Staubli VAL3: onEnterEvent.pgx

program onEnterEvent()
  local num i
  local num l_nIndex
  local string l_sItem[2]
  local num l_nResult
  local string l_sMessage
begin
  pub:libLoad("Disk://page/page_editTraj")
  call pub:main()
end
